TYPE WcStateBase_A2171C4E :
STRUCT
END_STRUCT
END_TYPE

(* stored: Version 1.2.0.0, ProductVersion 3.1.4024.9
   DUT WcStateBase_A2171C4E: Id {36551c0d-cfa8-4550-b14f-ac2cba101b6c} *)
